TYPE DUT_MotionStage_Extras :
STRUCT
    fVisuStep: LREAL;
    bVisuLowLim: BOOL;
    bVisuHighLim: BOOL;
END_STRUCT
END_TYPE

(* stored: Version 1.1.0.1, ProductVersion 3.1.4024.4
   DUT DUT_MotionStage_Extras: Id {1e6627e8-279b-4e38-87a2-ae79853e08df} *)
